FUNCTION_BLOCK animacao_icone_gerador (* Basic Function Block Type *)
  (* Standard: 61499-2 *)
  (* Version 0.0, 03/06/2026, Template *)
  PACKAGE Hidryco.HidrycoLib;
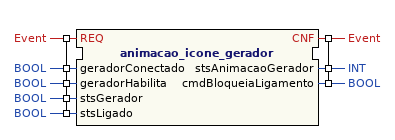
  EVENT_INPUT
    REQ WITH geradorConectado, geradorHabilita, stsGerador, stsLigado; (* Normal Execution Request *)
  END_EVENT
  EVENT_OUTPUT
    CNF WITH stsAnimacaoGerador, cmdBloqueiaLigamento; (* Execution Confirmation *)
  END_EVENT
  VAR_INPUT
    geradorConectado : BOOL;
    geradorHabilita : BOOL;
    stsGerador : BOOL; (* Status do Gerador ligado *)
    stsLigado : BOOL;
  END_VAR
  VAR_OUTPUT
    stsAnimacaoGerador : INT;
    cmdBloqueiaLigamento : BOOL;
  END_VAR
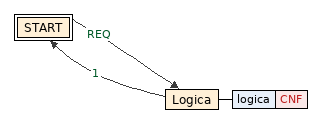
  EC_STATES
    START; (* Initial State *)
    Logica : logica -> CNF;
  END_STATES
  EC_TRANSITIONS
    START TO Logica := REQ;
    Logica TO START := 1;
  END_TRANSITIONS
  ALGORITHM logica IN ST:
// animação
IF NOT geradorConectado THEN
    stsAnimacaoGerador := 0;
ELSIF NOT geradorHabilita THEN
    stsAnimacaoGerador := 1;
ELSIF stsLigado AND stsGerador THEN
    stsAnimacaoGerador := 3;
ELSE
    stsAnimacaoGerador := 2;
END_IF;

// bloqueia o ligamento sempre que não há gerador disponível e habilitado
cmdBloqueiaLigamento := stsGerador AND NOT (geradorConectado AND geradorHabilita);

;
  END_ALGORITHM
END_FUNCTION_BLOCK
